Staubli VAL3: getProgItem.pgx

public program getProgItem(progItem& x_pProgItem, string x_sName)
  local num l_nResult
  local string l_sPath
  local string l_sName
begin
  if isDefined(saveProg:pProg[x_sName])
    // give back
    x_pProgItem=saveProg:pProg[x_sName]
    x_pProgItem.sID=x_sName
  else
    // TODO
    popUpMsg("PROG: "+x_sName+" NOT FOUND ")
    x_pProgItem.sID=""
  endIf
end
